FUNCTION_BLOCK FB_MyFB
VAR_INPUT
END_VAR
VAR_OUTPUT
END_VAR
VAR
END_VAR

END_FUNCTION_BLOCK

(* stored: Version 1.1.0.1
   POU FB_MyFB: Id {8d259eaa-df04-4172-ab05-ec30e9b40def}, SpecialFunc None *)
